// TIA Portal project "ISA_P3" (V16)

(* hardware
DEVICE "S7-1200 station_1"  S7-1200 Station
   slot 0: "Rack_0"  S7-1200 Rack  Rack  V1.0
   slot 1: "PLC_1"  CPU 1215C DC/DC/DC  6ES7 215-1AG40-0XB0  V4.4
   slot 2: "AI 4x13BIT/AQ 2x14BIT_1"  SM 1234 AI4/AQ2  6ES7 234-4HE30-0XB0  V1.0
DEVICE "PC-System_1"  SIMATIC PC station
   slot 0: "Estación PC SIMATIC"  Rail  SIMATIC PC-Station  V1.0
      slot 125: "Stationmanager"  Station_Manager  V6.0.4
   slot 1: "HMI_RT_1"  WinCC RT Advanced  6AV2 104-0xxxx-xxxx  16.0.0.0
      slot 33792: "Interfaz del equipo"  Host interface
   slot 2: "IE general_1"  IE General  IE_CP  V8.2.0
*)

// ===== PLC "PLC_1"  CPU 1215C DC/DC/DC =====

VAR_GLOBAL   // PLC tag table "Tabla de variables estándar"
   "raw_weight" AT %IW96 : Int;
   "raw_intensity" AT %IW98 : Int;
   "lamp" AT %QW96 : Int;
   "S1" AT %I0.0 : Bool;
END_VAR

DATA_BLOCK "Variable"   // DB1
{ S7_Optimized_Access := 'TRUE' }
VERSION : 0.1
   VAR
      norm_weight : Real;
      weight : Real;
      norm_intensity : Real;
      intensity : Int;
      raw_time : DTL;
      norm_time : Real;
      "time" : Int;
      modos : Int;
      lamp_variable : Real;
      lamp_norm : Real;
      lamp : Int;
      "on/off" : Bool;
      state : Bool;
      flanco_S1 : Bool;
      time_error : Int;
   END_VAR
BEGIN
END_DATA_BLOCK

ORGANIZATION_BLOCK "Scales"   // OB1, LAD, ProgramCycle
TITLE = "Main Program Sweep (Cycle)"
{ S7_Optimized_Access := 'TRUE' }
VERSION : 0.1
   VAR_INPUT
      Initial_Call : Bool;   // Initial call of this OB
      Remanence : Bool;   // =True, if remanent data are available
   END_VAR
BEGIN

REGION Network 1: Escalado de la célula de carga
   // El acondicionador de la célula de carga entrega una señal de 0 a 20mA para un rango de entrada de 0 a 3843.5kg, que equivale a una señal de 0 a 27648 bits.
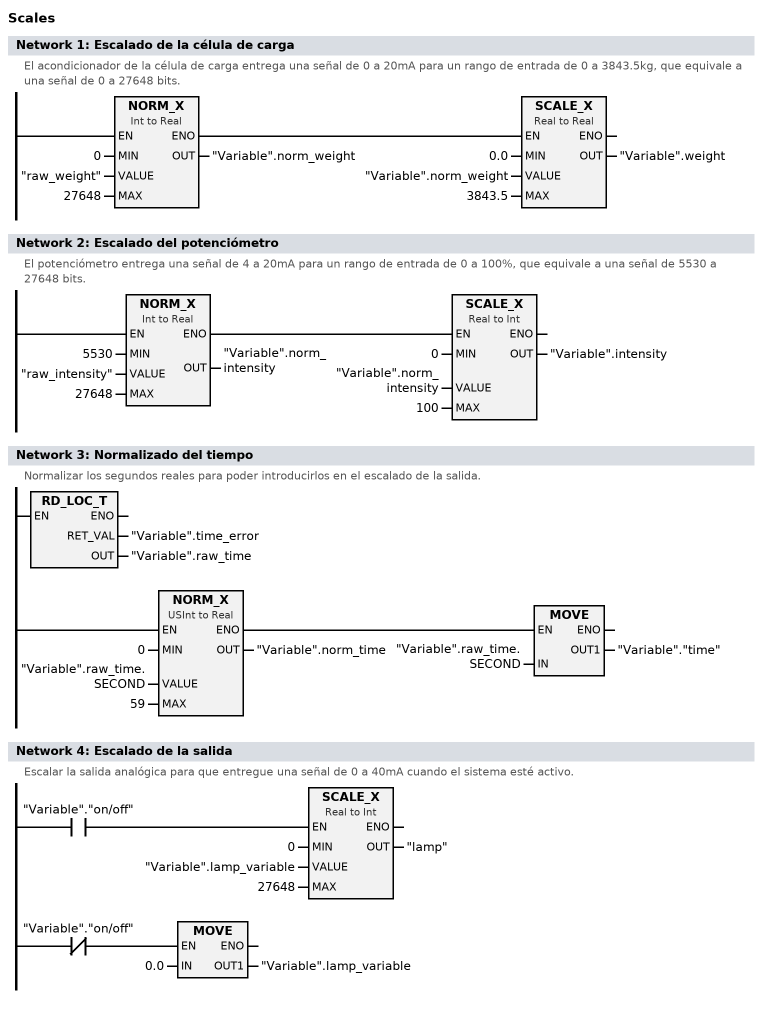
   RUNG wire#powerrail
      { S7_Templates := "[SrcType := Int, DestType := Real]" } Normalize(min := 0, value := "raw_weight", max := 27648, out => "Variable".norm_weight)
      { S7_Templates := "[SrcType := Real, DestType := Real]" } Scale(min := 0.0, value := "Variable".norm_weight, max := 3843.5, out => "Variable".weight)
   END_RUNG
   // the same network as SCL:
   "Variable".norm_weight := NORM_X(MIN := 0, VALUE := "raw_weight", MAX := 27648);
   "Variable".weight := SCALE_X(MIN := 0.0, VALUE := "Variable".norm_weight, MAX := 3843.5);
END_REGION

REGION Network 2: Escalado del potenciómetro
   // El potenciómetro entrega una señal de 4 a 20mA para un rango de entrada de 0 a 100%, que equivale a una señal de 5530 a 27648 bits.
   RUNG wire#powerrail
      { S7_Templates := "[SrcType := Int, DestType := Real]" } Normalize(min := 5530, value := "raw_intensity", max := 27648, out => "Variable".norm_intensity)
      { S7_Templates := "[SrcType := Real, DestType := Int]" } Scale(min := 0, value := "Variable".norm_intensity, max := 100, out => "Variable".intensity)
   END_RUNG
   // the same network as SCL:
   "Variable".norm_intensity := NORM_X(MIN := 5530, VALUE := "raw_intensity", MAX := 27648);
   "Variable".intensity := SCALE_X(MIN := 0, VALUE := "Variable".norm_intensity, MAX := 100);
END_REGION

REGION Network 3: Normalizado del tiempo
   // Normalizar los segundos reales para poder introducirlos en el escalado de la salida.
   "Variable".time_error := RD_LOC_T(OUT => "Variable".raw_time);
   "Variable".norm_time := NORM_X(MIN := 0, VALUE := "Variable".raw_time.SECOND, MAX := 59);
   "Variable"."time" := "Variable".raw_time.SECOND;
END_REGION

REGION Network 4: Escalado de la salida
   // Escalar la salida analógica para que entregue una señal de 0 a 40mA cuando el sistema esté activo.
   RUNG wire#powerrail
      Contact( "Variable"."on/off" )
      { S7_Templates := "[SrcType := Real, DestType := Int]" } Scale(min := 0, value := "Variable".lamp_variable, max := 27648, out => "lamp")
   END_RUNG
   RUNG wire#powerrail
      I_Contact( "Variable"."on/off" )
      Move(in := 0.0, out1 => "Variable".lamp_variable)
   END_RUNG
   // the same network as SCL:
   IF "Variable"."on/off" THEN
       "lamp" := SCALE_X(MIN := 0, VALUE := "Variable".lamp_variable, MAX := 27648);
   END_IF;
   IF NOT "Variable"."on/off" THEN "Variable".lamp_variable := 0.0; END_IF;
END_REGION
END_ORGANIZATION_BLOCK

ORGANIZATION_BLOCK "Main"   // OB123, LAD, ProgramCycle
TITLE = "Main Program Sweep (Cycle)"
{ S7_Optimized_Access := 'TRUE' }
VERSION : 0.1
   VAR_INPUT
      Initial_Call : Bool;   // Initial call of this OB
      Remanence : Bool;   // =True, if remanent data are available
   END_VAR
   VAR_TEMP   // added for the SCL form of the ladder/FBD networks
      _w1 : Bool;
   END_VAR
BEGIN

REGION Network 1: Telerruptor
   // Lógica de la función telerruptor del interruptor: Al pulsarse S1, si on/off estaba desactivada, la activará. De lo contrario, la desactivará.
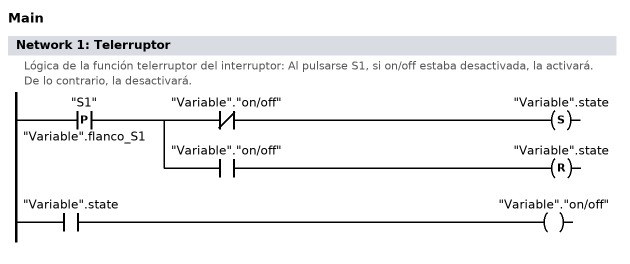
   RUNG wire#powerrail
      P_Contact(operand := "S1", bit := "Variable".flanco_S1)
      wire#w1
      I_Contact( "Variable"."on/off" )
      S_Coil( "Variable".state )
   END_RUNG
   RUNG wire#w1
      Contact( "Variable"."on/off" )
      R_Coil( "Variable".state )
   END_RUNG
   RUNG wire#powerrail
      Contact( "Variable".state )
      Coil( "Variable"."on/off" )
   END_RUNG
   // the same network as SCL:
   #_w1 := "S1" AND NOT "Variable".flanco_S1;   // rising edge of "S1"
   "Variable".flanco_S1 := "S1";
   IF #_w1 AND NOT "Variable"."on/off" THEN "Variable".state := TRUE; END_IF;
   IF #_w1 AND "Variable"."on/off" THEN "Variable".state := FALSE; END_IF;
   "Variable"."on/off" := "Variable".state;
END_REGION

REGION Network 2 (SCL): Conmutación de variables de salida
   // Según el modo seleccionado en SCADA, enviar una de las 3 señales normalizadas que pueden variar la salida a la variable que alimenta el escalado de dicha salida.
   // Se invierte la variable del peso para que el peso en la célula de carga sea inversamente proporcional a la intensidad con la que brilla la bombilla.
   IF "Variable".modos = 0 THEN
       "Variable".lamp_variable := "Variable".norm_intensity;
   ELSIF "Variable".modos = 1 THEN
       "Variable".lamp_variable := 1.0 - "Variable".norm_weight;
   ELSE
       "Variable".lamp_variable := "Variable".norm_time;
   END_IF;
END_REGION
END_ORGANIZATION_BLOCK

(* ===== HMI "HMI_RT_1" =====
connection "HMI_Conexión_1": ETHERNET, S7_1200_OMS

HMI tags "Tabla de variables estándar"
   "Variable_modos" : Int = PLC Variable.modos, 1 s
   "Variable_weight" : Real = PLC Variable.weight, 1 s
   "Variable_intensity" : Int = PLC Variable.intensity, 1 s
   "Variable_norm_time" : Real = PLC Variable.norm_time, 1 s
   "Variable_time" : Int = PLC Variable.time, 1 s

text list "Lista de textos_1": 0 'Manual'; 1 'Peso'; 2 'Tiempo'

screen "recor" 800x600
   SymbolicIOField "Campo ES simbólico_1" at 313,205 size 161x70; TextOff '0'; TextOn '1'; TextList "Lista de textos_1"
      ProcessValue <- "Variable_modos"
   IOField "Campo ES_1" at 95,353 size 96x32; FormatPattern 999
      ProcessValue <- "Variable_intensity"
   IOField "Campo ES_2" at 333,353 size 96x32; FormatPattern 9999.9
      ProcessValue <- "Variable_weight"
   IOField "Campo ES_3" at 571,353 size 96x32; FormatPattern 99
      ProcessValue <- "Variable_time"
   TextField "Campo de texto_1" at 96,307 size 73x22; Text 'Intensity'
   TextField "Campo de texto_2" at 334,306 size 58x22; Text 'Weight'
   TextField "Campo de texto_3" at 569,308 size 67x22; Text 'Seconds'
*)